// TIA Portal V19 export
FUNCTION "A0304_Navetta_CALL" : Void   // FC147, LAD
// stored: SetENOAutomatically false
BEGIN

REGION Network 1: <<< LATO TESTA >>>
END_REGION

REGION Network 2: DataIn - Ax
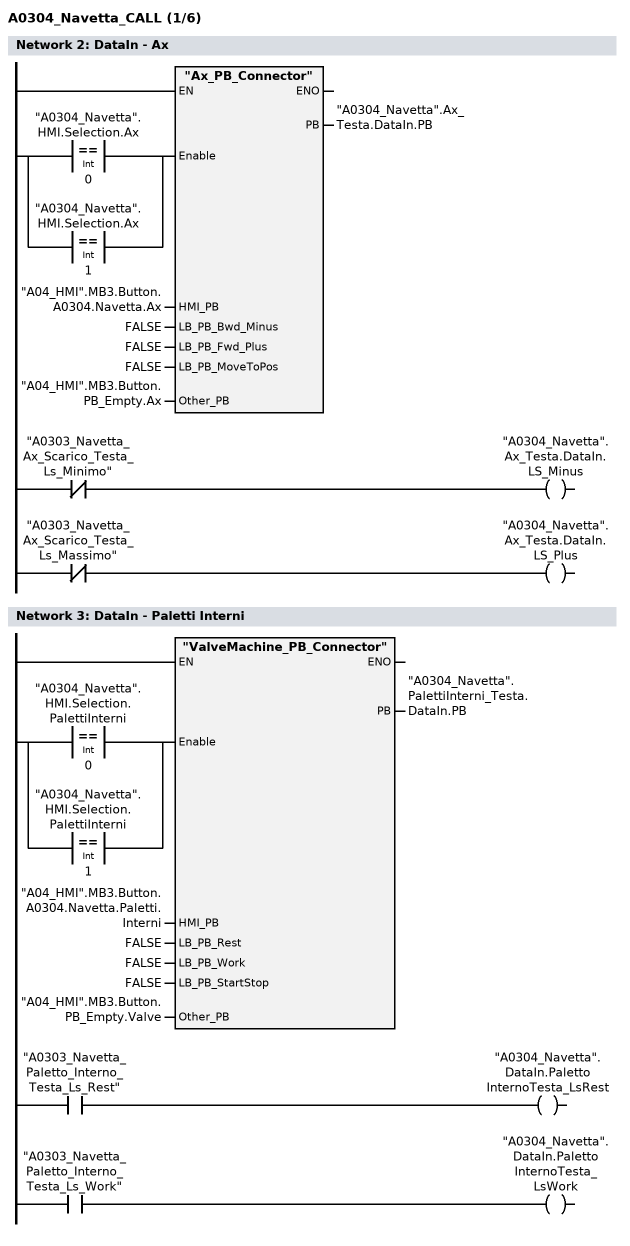
   RUNG wire#powerrail
      "Ax_PB_Connector"(Enable := wire#w1, HMI_PB := "A04_HMI".MB3.Button.A0304.Navetta.Ax, LB_PB_Bwd_Minus := FALSE, LB_PB_Fwd_Plus := FALSE, LB_PB_MoveToPos := FALSE, Other_PB := "A04_HMI".MB3.Button.PB_Empty.Ax, PB => "A0304_Navetta".Ax_Testa.DataIn.PB)
   END_RUNG
   RUNG wire#powerrail
      { S7_Templates := "SrcType := Int" } EQ_Contact(in1 := "A0304_Navetta".HMI.Selection.Ax, in2 := 0)
   END_RUNG wire#w1
   RUNG wire#powerrail
      { S7_Templates := "SrcType := Int" } EQ_Contact(in1 := "A0304_Navetta".HMI.Selection.Ax, in2 := 1)
   END_RUNG wire#w1
   RUNG wire#powerrail
      I_Contact( "A0303_Navetta_Ax_Scarico_Testa_Ls_Minimo" )
      Coil( "A0304_Navetta".Ax_Testa.DataIn.LS_Minus )
   END_RUNG
   RUNG wire#powerrail
      I_Contact( "A0303_Navetta_Ax_Scarico_Testa_Ls_Massimo" )
      Coil( "A0304_Navetta".Ax_Testa.DataIn.LS_Plus )
   END_RUNG
   // the same network as SCL:
   "Ax_PB_Connector"(Enable := ("A0304_Navetta".HMI.Selection.Ax = 0) OR ("A0304_Navetta".HMI.Selection.Ax = 1),
                     HMI_PB := "A04_HMI".MB3.Button.A0304.Navetta.Ax,
                     LB_PB_Bwd_Minus := FALSE,
                     LB_PB_Fwd_Plus := FALSE,
                     LB_PB_MoveToPos := FALSE,
                     Other_PB := "A04_HMI".MB3.Button.PB_Empty.Ax,
                     PB => "A0304_Navetta".Ax_Testa.DataIn.PB);
   "A0304_Navetta".Ax_Testa.DataIn.LS_Minus := NOT "A0303_Navetta_Ax_Scarico_Testa_Ls_Minimo";
   "A0304_Navetta".Ax_Testa.DataIn.LS_Plus := NOT "A0303_Navetta_Ax_Scarico_Testa_Ls_Massimo";
END_REGION

REGION Network 3: DataIn - Paletti Interni
   RUNG wire#powerrail
      "ValveMachine_PB_Connector"(Enable := wire#w1, HMI_PB := "A04_HMI".MB3.Button.A0304.Navetta.Paletti.Interni, LB_PB_Rest := FALSE, LB_PB_Work := FALSE, LB_PB_StartStop := FALSE, Other_PB := "A04_HMI".MB3.Button.PB_Empty.Valve, PB => "A0304_Navetta".PalettiInterni_Testa.DataIn.PB)
   END_RUNG
   RUNG wire#powerrail
      { S7_Templates := "SrcType := Int" } EQ_Contact(in1 := "A0304_Navetta".HMI.Selection.PalettiInterni, in2 := 0)
   END_RUNG wire#w1
   RUNG wire#powerrail
      { S7_Templates := "SrcType := Int" } EQ_Contact(in1 := "A0304_Navetta".HMI.Selection.PalettiInterni, in2 := 1)
   END_RUNG wire#w1
   RUNG wire#powerrail
      Contact( "A0303_Navetta_Paletto_Interno_Testa_Ls_Rest" )
      Coil( "A0304_Navetta".DataIn.PalettoInternoTesta_LsRest )
   END_RUNG
   RUNG wire#powerrail
      Contact( "A0303_Navetta_Paletto_Interno_Testa_Ls_Work" )
      Coil( "A0304_Navetta".DataIn.PalettoInternoTesta_LsWork )
   END_RUNG
   // the same network as SCL:
   "ValveMachine_PB_Connector"(Enable := ("A0304_Navetta".HMI.Selection.PalettiInterni = 0) OR ("A0304_Navetta".HMI.Selection.PalettiInterni = 1),
                           HMI_PB := "A04_HMI".MB3.Button.A0304.Navetta.Paletti.Interni,
                           LB_PB_Rest := FALSE,
                           LB_PB_Work := FALSE,
                           LB_PB_StartStop := FALSE,
                           Other_PB := "A04_HMI".MB3.Button.PB_Empty.Valve,
                           PB => "A0304_Navetta".PalettiInterni_Testa.DataIn.PB);
   "A0304_Navetta".DataIn.PalettoInternoTesta_LsRest := "A0303_Navetta_Paletto_Interno_Testa_Ls_Rest";
   "A0304_Navetta".DataIn.PalettoInternoTesta_LsWork := "A0303_Navetta_Paletto_Interno_Testa_Ls_Work";
END_REGION

REGION Network 4: DataIn - Paletti Esterni
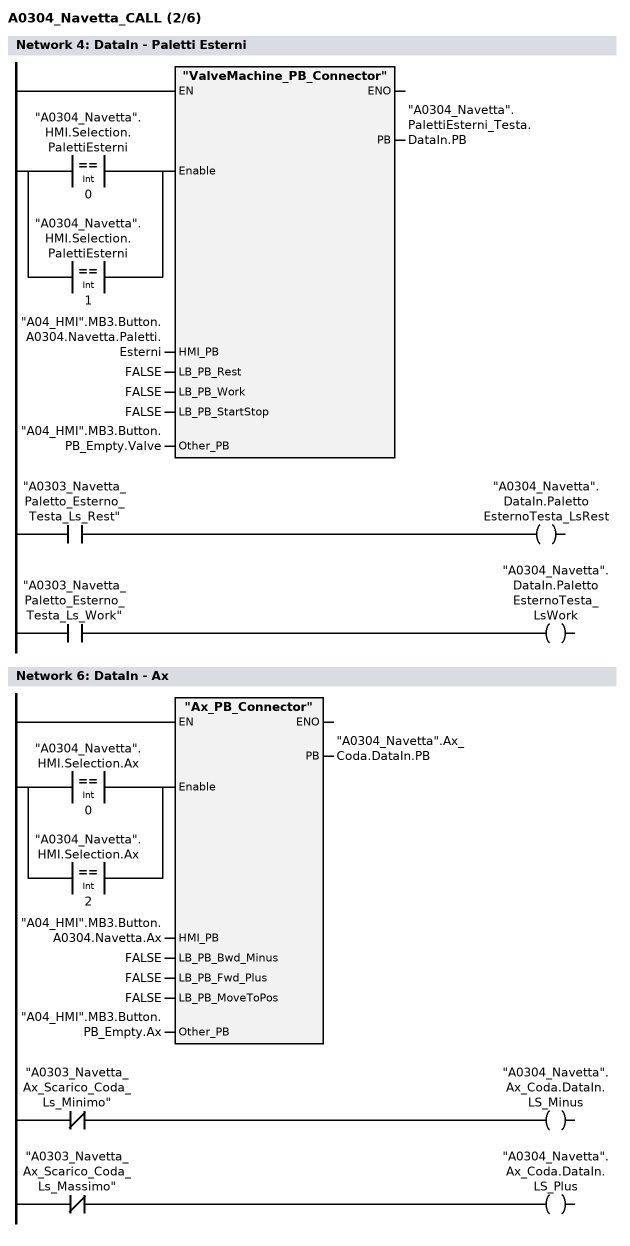
   RUNG wire#powerrail
      "ValveMachine_PB_Connector"(Enable := wire#w1, HMI_PB := "A04_HMI".MB3.Button.A0304.Navetta.Paletti.Esterni, LB_PB_Rest := FALSE, LB_PB_Work := FALSE, LB_PB_StartStop := FALSE, Other_PB := "A04_HMI".MB3.Button.PB_Empty.Valve, PB => "A0304_Navetta".PalettiEsterni_Testa.DataIn.PB)
   END_RUNG
   RUNG wire#powerrail
      { S7_Templates := "SrcType := Int" } EQ_Contact(in1 := "A0304_Navetta".HMI.Selection.PalettiEsterni, in2 := 0)
   END_RUNG wire#w1
   RUNG wire#powerrail
      { S7_Templates := "SrcType := Int" } EQ_Contact(in1 := "A0304_Navetta".HMI.Selection.PalettiEsterni, in2 := 1)
   END_RUNG wire#w1
   RUNG wire#powerrail
      Contact( "A0303_Navetta_Paletto_Esterno_Testa_Ls_Rest" )
      Coil( "A0304_Navetta".DataIn.PalettoEsternoTesta_LsRest )
   END_RUNG
   RUNG wire#powerrail
      Contact( "A0303_Navetta_Paletto_Esterno_Testa_Ls_Work" )
      Coil( "A0304_Navetta".DataIn.PalettoEsternoTesta_LsWork )
   END_RUNG
   // the same network as SCL:
   "ValveMachine_PB_Connector"(Enable := ("A0304_Navetta".HMI.Selection.PalettiEsterni = 0) OR ("A0304_Navetta".HMI.Selection.PalettiEsterni = 1),
                           HMI_PB := "A04_HMI".MB3.Button.A0304.Navetta.Paletti.Esterni,
                           LB_PB_Rest := FALSE,
                           LB_PB_Work := FALSE,
                           LB_PB_StartStop := FALSE,
                           Other_PB := "A04_HMI".MB3.Button.PB_Empty.Valve,
                           PB => "A0304_Navetta".PalettiEsterni_Testa.DataIn.PB);
   "A0304_Navetta".DataIn.PalettoEsternoTesta_LsRest := "A0303_Navetta_Paletto_Esterno_Testa_Ls_Rest";
   "A0304_Navetta".DataIn.PalettoEsternoTesta_LsWork := "A0303_Navetta_Paletto_Esterno_Testa_Ls_Work";
END_REGION

REGION Network 5: <<< LATO CODA >>>
END_REGION

REGION Network 6: DataIn - Ax
   RUNG wire#powerrail
      "Ax_PB_Connector"(Enable := wire#w1, HMI_PB := "A04_HMI".MB3.Button.A0304.Navetta.Ax, LB_PB_Bwd_Minus := FALSE, LB_PB_Fwd_Plus := FALSE, LB_PB_MoveToPos := FALSE, Other_PB := "A04_HMI".MB3.Button.PB_Empty.Ax, PB => "A0304_Navetta".Ax_Coda.DataIn.PB)
   END_RUNG
   RUNG wire#powerrail
      { S7_Templates := "SrcType := Int" } EQ_Contact(in1 := "A0304_Navetta".HMI.Selection.Ax, in2 := 0)
   END_RUNG wire#w1
   RUNG wire#powerrail
      { S7_Templates := "SrcType := Int" } EQ_Contact(in1 := "A0304_Navetta".HMI.Selection.Ax, in2 := 2)
   END_RUNG wire#w1
   RUNG wire#powerrail
      I_Contact( "A0303_Navetta_Ax_Scarico_Coda_Ls_Minimo" )
      Coil( "A0304_Navetta".Ax_Coda.DataIn.LS_Minus )
   END_RUNG
   RUNG wire#powerrail
      I_Contact( "A0303_Navetta_Ax_Scarico_Coda_Ls_Massimo" )
      Coil( "A0304_Navetta".Ax_Coda.DataIn.LS_Plus )
   END_RUNG
   // the same network as SCL:
   "Ax_PB_Connector"(Enable := ("A0304_Navetta".HMI.Selection.Ax = 0) OR ("A0304_Navetta".HMI.Selection.Ax = 2),
                     HMI_PB := "A04_HMI".MB3.Button.A0304.Navetta.Ax,
                     LB_PB_Bwd_Minus := FALSE,
                     LB_PB_Fwd_Plus := FALSE,
                     LB_PB_MoveToPos := FALSE,
                     Other_PB := "A04_HMI".MB3.Button.PB_Empty.Ax,
                     PB => "A0304_Navetta".Ax_Coda.DataIn.PB);
   "A0304_Navetta".Ax_Coda.DataIn.LS_Minus := NOT "A0303_Navetta_Ax_Scarico_Coda_Ls_Minimo";
   "A0304_Navetta".Ax_Coda.DataIn.LS_Plus := NOT "A0303_Navetta_Ax_Scarico_Coda_Ls_Massimo";
END_REGION

REGION Network 7: DataIn - Paletti Interni
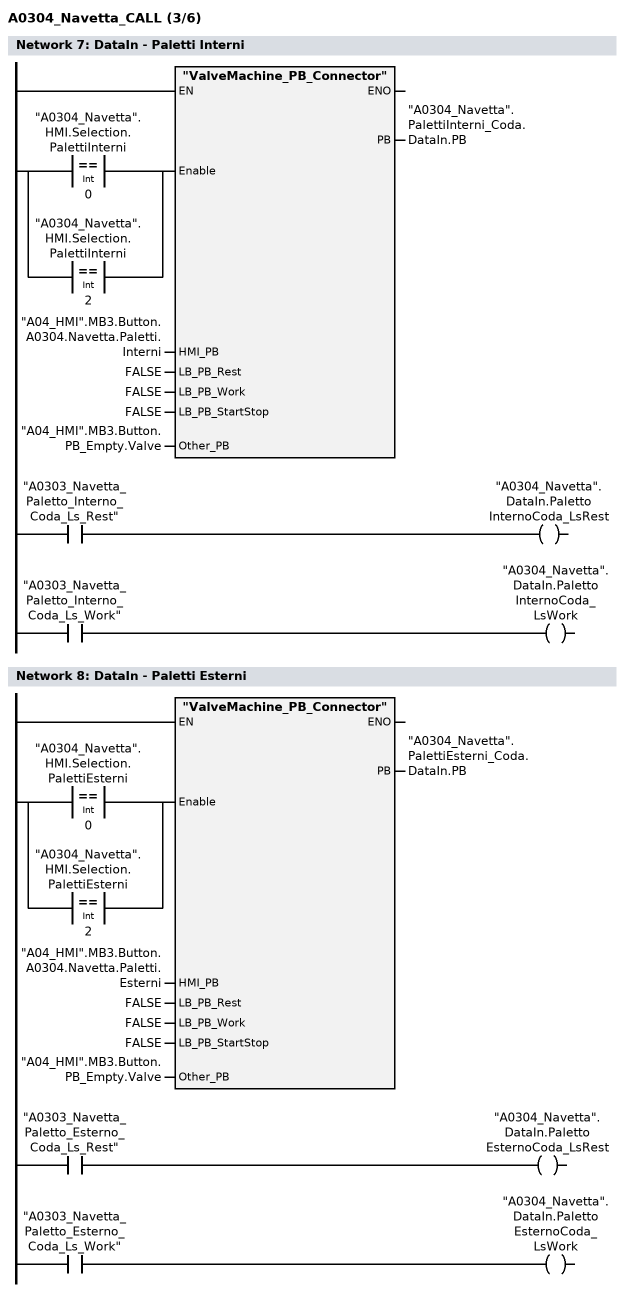
   RUNG wire#powerrail
      "ValveMachine_PB_Connector"(Enable := wire#w1, HMI_PB := "A04_HMI".MB3.Button.A0304.Navetta.Paletti.Interni, LB_PB_Rest := FALSE, LB_PB_Work := FALSE, LB_PB_StartStop := FALSE, Other_PB := "A04_HMI".MB3.Button.PB_Empty.Valve, PB => "A0304_Navetta".PalettiInterni_Coda.DataIn.PB)
   END_RUNG
   RUNG wire#powerrail
      { S7_Templates := "SrcType := Int" } EQ_Contact(in1 := "A0304_Navetta".HMI.Selection.PalettiInterni, in2 := 0)
   END_RUNG wire#w1
   RUNG wire#powerrail
      { S7_Templates := "SrcType := Int" } EQ_Contact(in1 := "A0304_Navetta".HMI.Selection.PalettiInterni, in2 := 2)
   END_RUNG wire#w1
   RUNG wire#powerrail
      Contact( "A0303_Navetta_Paletto_Interno_Coda_Ls_Rest" )
      Coil( "A0304_Navetta".DataIn.PalettoInternoCoda_LsRest )
   END_RUNG
   RUNG wire#powerrail
      Contact( "A0303_Navetta_Paletto_Interno_Coda_Ls_Work" )
      Coil( "A0304_Navetta".DataIn.PalettoInternoCoda_LsWork )
   END_RUNG
   // the same network as SCL:
   "ValveMachine_PB_Connector"(Enable := ("A0304_Navetta".HMI.Selection.PalettiInterni = 0) OR ("A0304_Navetta".HMI.Selection.PalettiInterni = 2),
                           HMI_PB := "A04_HMI".MB3.Button.A0304.Navetta.Paletti.Interni,
                           LB_PB_Rest := FALSE,
                           LB_PB_Work := FALSE,
                           LB_PB_StartStop := FALSE,
                           Other_PB := "A04_HMI".MB3.Button.PB_Empty.Valve,
                           PB => "A0304_Navetta".PalettiInterni_Coda.DataIn.PB);
   "A0304_Navetta".DataIn.PalettoInternoCoda_LsRest := "A0303_Navetta_Paletto_Interno_Coda_Ls_Rest";
   "A0304_Navetta".DataIn.PalettoInternoCoda_LsWork := "A0303_Navetta_Paletto_Interno_Coda_Ls_Work";
END_REGION

REGION Network 8: DataIn - Paletti Esterni
   RUNG wire#powerrail
      "ValveMachine_PB_Connector"(Enable := wire#w1, HMI_PB := "A04_HMI".MB3.Button.A0304.Navetta.Paletti.Esterni, LB_PB_Rest := FALSE, LB_PB_Work := FALSE, LB_PB_StartStop := FALSE, Other_PB := "A04_HMI".MB3.Button.PB_Empty.Valve, PB => "A0304_Navetta".PalettiEsterni_Coda.DataIn.PB)
   END_RUNG
   RUNG wire#powerrail
      { S7_Templates := "SrcType := Int" } EQ_Contact(in1 := "A0304_Navetta".HMI.Selection.PalettiEsterni, in2 := 0)
   END_RUNG wire#w1
   RUNG wire#powerrail
      { S7_Templates := "SrcType := Int" } EQ_Contact(in1 := "A0304_Navetta".HMI.Selection.PalettiEsterni, in2 := 2)
   END_RUNG wire#w1
   RUNG wire#powerrail
      Contact( "A0303_Navetta_Paletto_Esterno_Coda_Ls_Rest" )
      Coil( "A0304_Navetta".DataIn.PalettoEsternoCoda_LsRest )
   END_RUNG
   RUNG wire#powerrail
      Contact( "A0303_Navetta_Paletto_Esterno_Coda_Ls_Work" )
      Coil( "A0304_Navetta".DataIn.PalettoEsternoCoda_LsWork )
   END_RUNG
   // the same network as SCL:
   "ValveMachine_PB_Connector"(Enable := ("A0304_Navetta".HMI.Selection.PalettiEsterni = 0) OR ("A0304_Navetta".HMI.Selection.PalettiEsterni = 2),
                           HMI_PB := "A04_HMI".MB3.Button.A0304.Navetta.Paletti.Esterni,
                           LB_PB_Rest := FALSE,
                           LB_PB_Work := FALSE,
                           LB_PB_StartStop := FALSE,
                           Other_PB := "A04_HMI".MB3.Button.PB_Empty.Valve,
                           PB => "A0304_Navetta".PalettiEsterni_Coda.DataIn.PB);
   "A0304_Navetta".DataIn.PalettoEsternoCoda_LsRest := "A0303_Navetta_Paletto_Esterno_Coda_Ls_Rest";
   "A0304_Navetta".DataIn.PalettoEsternoCoda_LsWork := "A0303_Navetta_Paletto_Esterno_Coda_Ls_Work";
END_REGION

REGION Network 10: DataIn - Material Presence
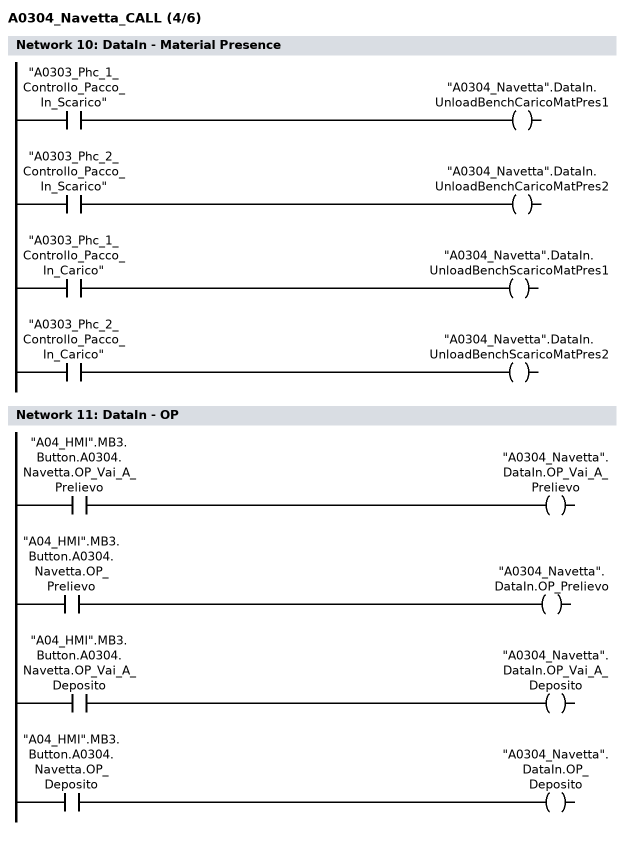
   RUNG wire#powerrail
      Contact( "A0303_Phc_1_Controllo_Pacco_In_Scarico" )
      Coil( "A0304_Navetta".DataIn.UnloadBenchCaricoMatPres1 )
   END_RUNG
   RUNG wire#powerrail
      Contact( "A0303_Phc_2_Controllo_Pacco_In_Scarico" )
      Coil( "A0304_Navetta".DataIn.UnloadBenchCaricoMatPres2 )
   END_RUNG
   RUNG wire#powerrail
      Contact( "A0303_Phc_1_Controllo_Pacco_In_Carico" )
      Coil( "A0304_Navetta".DataIn.UnloadBenchScaricoMatPres1 )
   END_RUNG
   RUNG wire#powerrail
      Contact( "A0303_Phc_2_Controllo_Pacco_In_Carico" )
      Coil( "A0304_Navetta".DataIn.UnloadBenchScaricoMatPres2 )
   END_RUNG
   // the same network as SCL:
   "A0304_Navetta".DataIn.UnloadBenchCaricoMatPres1 := "A0303_Phc_1_Controllo_Pacco_In_Scarico";
   "A0304_Navetta".DataIn.UnloadBenchCaricoMatPres2 := "A0303_Phc_2_Controllo_Pacco_In_Scarico";
   "A0304_Navetta".DataIn.UnloadBenchScaricoMatPres1 := "A0303_Phc_1_Controllo_Pacco_In_Carico";
   "A0304_Navetta".DataIn.UnloadBenchScaricoMatPres2 := "A0303_Phc_2_Controllo_Pacco_In_Carico";
END_REGION

REGION Network 11: DataIn - OP
   RUNG wire#powerrail
      Contact( "A04_HMI".MB3.Button.A0304.Navetta.OP_Vai_A_Prelievo )
      Coil( "A0304_Navetta".DataIn.OP_Vai_A_Prelievo )
   END_RUNG
   RUNG wire#powerrail
      Contact( "A04_HMI".MB3.Button.A0304.Navetta.OP_Prelievo )
      Coil( "A0304_Navetta".DataIn.OP_Prelievo )
   END_RUNG
   RUNG wire#powerrail
      Contact( "A04_HMI".MB3.Button.A0304.Navetta.OP_Vai_A_Deposito )
      Coil( "A0304_Navetta".DataIn.OP_Vai_A_Deposito )
   END_RUNG
   RUNG wire#powerrail
      Contact( "A04_HMI".MB3.Button.A0304.Navetta.OP_Deposito )
      Coil( "A0304_Navetta".DataIn.OP_Deposito )
   END_RUNG
   // the same network as SCL:
   "A0304_Navetta".DataIn.OP_Vai_A_Prelievo := "A04_HMI".MB3.Button.A0304.Navetta.OP_Vai_A_Prelievo;
   "A0304_Navetta".DataIn.OP_Prelievo := "A04_HMI".MB3.Button.A0304.Navetta.OP_Prelievo;
   "A0304_Navetta".DataIn.OP_Vai_A_Deposito := "A04_HMI".MB3.Button.A0304.Navetta.OP_Vai_A_Deposito;
   "A0304_Navetta".DataIn.OP_Deposito := "A04_HMI".MB3.Button.A0304.Navetta.OP_Deposito;
END_REGION

REGION Network 13: CIn
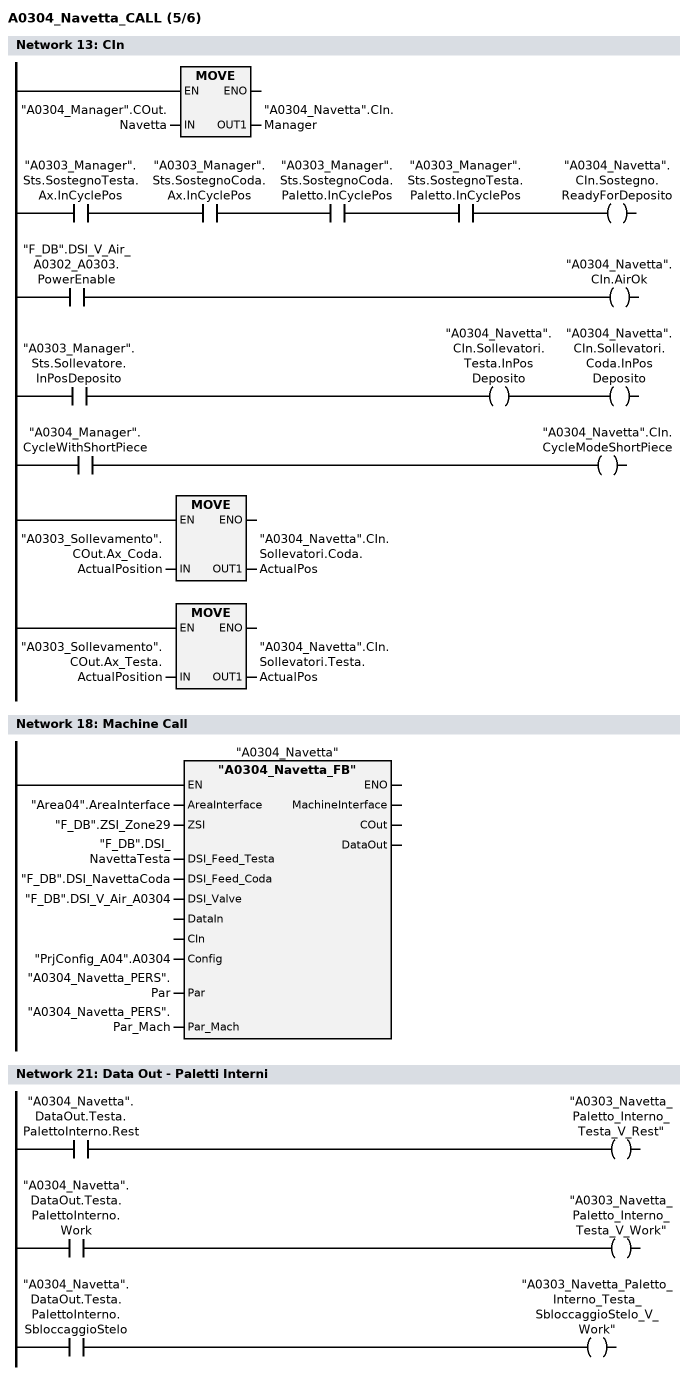
   RUNG wire#powerrail
      Move(in := "A0304_Manager".COut.Navetta, out1 => "A0304_Navetta".CIn.Manager)
   END_RUNG
   RUNG wire#powerrail
      Contact( "A0303_Manager".Sts.SostegnoTesta.Ax.InCyclePos )
      Contact( "A0303_Manager".Sts.SostegnoCoda.Ax.InCyclePos )
      Contact( "A0303_Manager".Sts.SostegnoCoda.Paletto.InCyclePos )
      Contact( "A0303_Manager".Sts.SostegnoTesta.Paletto.InCyclePos )
      Coil( "A0304_Navetta".CIn.Sostegno.ReadyForDeposito )
   END_RUNG
   RUNG wire#powerrail
      Contact( "F_DB".DSI_V_Air_A0302_A0303.PowerEnable )
      Coil( "A0304_Navetta".CIn.AirOk )
   END_RUNG
   RUNG wire#powerrail
      Contact( "A0303_Manager".Sts.Sollevatore.InPosDeposito )
      Coil( "A0304_Navetta".CIn.Sollevatori.Testa.InPosDeposito )
      Coil( "A0304_Navetta".CIn.Sollevatori.Coda.InPosDeposito )
   END_RUNG
   RUNG wire#powerrail
      Contact( "A0304_Manager".CycleWithShortPiece )
      Coil( "A0304_Navetta".CIn.CycleModeShortPiece )
   END_RUNG
   RUNG wire#powerrail
      Move(in := "A0303_Sollevamento".COut.Ax_Coda.ActualPosition, out1 => "A0304_Navetta".CIn.Sollevatori.Coda.ActualPos)
   END_RUNG
   RUNG wire#powerrail
      Move(in := "A0303_Sollevamento".COut.Ax_Testa.ActualPosition, out1 => "A0304_Navetta".CIn.Sollevatori.Testa.ActualPos)
   END_RUNG
   // the same network as SCL:
   "A0304_Navetta".CIn.Manager := "A0304_Manager".COut.Navetta;
   "A0304_Navetta".CIn.Sostegno.ReadyForDeposito := "A0303_Manager".Sts.SostegnoTesta.Ax.InCyclePos AND "A0303_Manager".Sts.SostegnoCoda.Ax.InCyclePos AND "A0303_Manager".Sts.SostegnoCoda.Paletto.InCyclePos AND "A0303_Manager".Sts.SostegnoTesta.Paletto.InCyclePos;
   "A0304_Navetta".CIn.AirOk := "F_DB".DSI_V_Air_A0302_A0303.PowerEnable;
   "A0304_Navetta".CIn.Sollevatori.Testa.InPosDeposito := "A0303_Manager".Sts.Sollevatore.InPosDeposito;
   "A0304_Navetta".CIn.Sollevatori.Coda.InPosDeposito := "A0303_Manager".Sts.Sollevatore.InPosDeposito;
   "A0304_Navetta".CIn.CycleModeShortPiece := "A0304_Manager".CycleWithShortPiece;
   "A0304_Navetta".CIn.Sollevatori.Coda.ActualPos := "A0303_Sollevamento".COut.Ax_Coda.ActualPosition;
   "A0304_Navetta".CIn.Sollevatori.Testa.ActualPos := "A0303_Sollevamento".COut.Ax_Testa.ActualPosition;
END_REGION

REGION Network 14: >
END_REGION

REGION Network 15 (SCL): Drive
   "A0304_Navetta".Ax_Testa.Drive.Infeed_ON := "Areas_ITF".AG.Infeed_Running;
   "A0304_Navetta".Ax_Testa.Drive.AccessPoint := "HW_Const_Values".CU8_PN_615A1_ModuleAccessPoint;
   "A0304_Navetta".Ax_Testa.Drive.AxisID := "CU8_ID_4_2430A1_1_2430M1";
   "A0304_Navetta".Ax_Testa.Drive.TokenChain := "TOKENCHAIN_CU8";

   "A0304_Navetta".Ax_Coda.Drive.Infeed_ON := "Areas_ITF".AG.Infeed_Running;
   "A0304_Navetta".Ax_Coda.Drive.AccessPoint := "HW_Const_Values".CU8_PN_615A1_ModuleAccessPoint;
   "A0304_Navetta".Ax_Coda.Drive.AxisID := "CU8_ID_5_2430A1_2_2460M1";
   "A0304_Navetta".Ax_Coda.Drive.TokenChain :=  "TOKENCHAIN_CU8";
END_REGION

REGION Network 16 (SCL): HW ID
   "A0304_Navetta".Ax_Testa.HW_ID_TEL1 := "HW_Const_Values".CU8_PN_2430A1_1_Standard_telegram_1;
   "A0304_Navetta".Enc_Testa.HW_IO := "HW_Const_Values".HW_2434P1_Telegram_81_DI_DO;

   "A0304_Navetta".Ax_Coda.HW_ID_TEL1 := "HW_Const_Values".CU8_PN_2430A1_2_Standard_telegram_1;
   "A0304_Navetta".Enc_Coda.HW_IO := "HW_Const_Values".HW_2464P1_Telegram_81_DI_DO;
END_REGION

REGION Network 17: >
END_REGION

REGION Network 18: Machine Call
   RUNG wire#powerrail
      "A0304_Navetta"(AreaInterface := "Area04".AreaInterface, ZSI := "F_DB".ZSI_Zone29, DSI_Feed_Testa := "F_DB".DSI_NavettaTesta, DSI_Feed_Coda := "F_DB".DSI_NavettaCoda, DSI_Valve := "F_DB".DSI_V_Air_A0304, DataIn :=, CIn :=, Config := "PrjConfig_A04".A0304, Par := "A0304_Navetta_PERS".Par, Par_Mach := "A0304_Navetta_PERS".Par_Mach, MachineInterface =>, COut =>, DataOut =>)
   END_RUNG
   // the same network as SCL:
   "A0304_Navetta"(AreaInterface := "Area04".AreaInterface,   // "A0304_Navetta_FB"
                   ZSI := "F_DB".ZSI_Zone29,
                   DSI_Feed_Testa := "F_DB".DSI_NavettaTesta,
                   DSI_Feed_Coda := "F_DB".DSI_NavettaCoda,
                   DSI_Valve := "F_DB".DSI_V_Air_A0304,
                   Config := "PrjConfig_A04".A0304,
                   Par := "A0304_Navetta_PERS".Par,
                   Par_Mach := "A0304_Navetta_PERS".Par_Mach);
END_REGION

REGION Network 20: <<< LATO TESTA >>>
END_REGION

REGION Network 21: Data Out - Paletti Interni
   RUNG wire#powerrail
      Contact( "A0304_Navetta".DataOut.Testa.PalettoInterno.Rest )
      Coil( "A0303_Navetta_Paletto_Interno_Testa_V_Rest" )
   END_RUNG
   RUNG wire#powerrail
      Contact( "A0304_Navetta".DataOut.Testa.PalettoInterno.Work )
      Coil( "A0303_Navetta_Paletto_Interno_Testa_V_Work" )
   END_RUNG
   RUNG wire#powerrail
      Contact( "A0304_Navetta".DataOut.Testa.PalettoInterno.SbloccaggioStelo )
      Coil( "A0303_Navetta_Paletto_Interno_Testa_SbloccaggioStelo_V_Work" )
   END_RUNG
   // the same network as SCL:
   "A0303_Navetta_Paletto_Interno_Testa_V_Rest" := "A0304_Navetta".DataOut.Testa.PalettoInterno.Rest;
   "A0303_Navetta_Paletto_Interno_Testa_V_Work" := "A0304_Navetta".DataOut.Testa.PalettoInterno.Work;
   "A0303_Navetta_Paletto_Interno_Testa_SbloccaggioStelo_V_Work" := "A0304_Navetta".DataOut.Testa.PalettoInterno.SbloccaggioStelo;
END_REGION

REGION Network 22: Data Out - Paletti Esterni
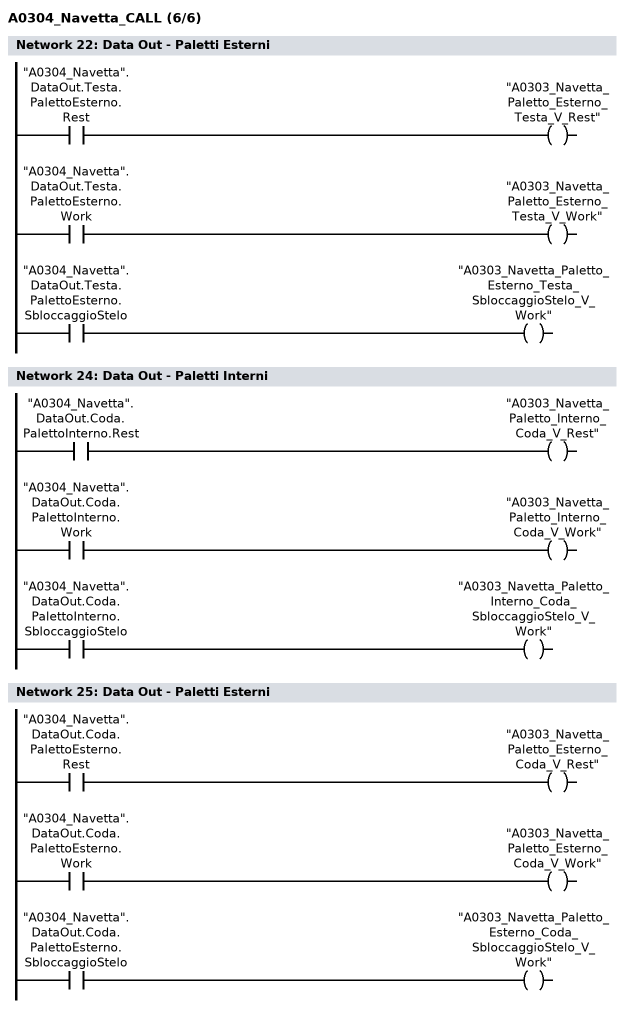
   RUNG wire#powerrail
      Contact( "A0304_Navetta".DataOut.Testa.PalettoEsterno.Rest )
      Coil( "A0303_Navetta_Paletto_Esterno_Testa_V_Rest" )
   END_RUNG
   RUNG wire#powerrail
      Contact( "A0304_Navetta".DataOut.Testa.PalettoEsterno.Work )
      Coil( "A0303_Navetta_Paletto_Esterno_Testa_V_Work" )
   END_RUNG
   RUNG wire#powerrail
      Contact( "A0304_Navetta".DataOut.Testa.PalettoEsterno.SbloccaggioStelo )
      Coil( "A0303_Navetta_Paletto_Esterno_Testa_SbloccaggioStelo_V_Work" )
   END_RUNG
   // the same network as SCL:
   "A0303_Navetta_Paletto_Esterno_Testa_V_Rest" := "A0304_Navetta".DataOut.Testa.PalettoEsterno.Rest;
   "A0303_Navetta_Paletto_Esterno_Testa_V_Work" := "A0304_Navetta".DataOut.Testa.PalettoEsterno.Work;
   "A0303_Navetta_Paletto_Esterno_Testa_SbloccaggioStelo_V_Work" := "A0304_Navetta".DataOut.Testa.PalettoEsterno.SbloccaggioStelo;
END_REGION

REGION Network 23: <<< LATO CODA >>>
END_REGION

REGION Network 24: Data Out - Paletti Interni
   RUNG wire#powerrail
      Contact( "A0304_Navetta".DataOut.Coda.PalettoInterno.Rest )
      Coil( "A0303_Navetta_Paletto_Interno_Coda_V_Rest" )
   END_RUNG
   RUNG wire#powerrail
      Contact( "A0304_Navetta".DataOut.Coda.PalettoInterno.Work )
      Coil( "A0303_Navetta_Paletto_Interno_Coda_V_Work" )
   END_RUNG
   RUNG wire#powerrail
      Contact( "A0304_Navetta".DataOut.Coda.PalettoInterno.SbloccaggioStelo )
      Coil( "A0303_Navetta_Paletto_Interno_Coda_SbloccaggioStelo_V_Work" )
   END_RUNG
   // the same network as SCL:
   "A0303_Navetta_Paletto_Interno_Coda_V_Rest" := "A0304_Navetta".DataOut.Coda.PalettoInterno.Rest;
   "A0303_Navetta_Paletto_Interno_Coda_V_Work" := "A0304_Navetta".DataOut.Coda.PalettoInterno.Work;
   "A0303_Navetta_Paletto_Interno_Coda_SbloccaggioStelo_V_Work" := "A0304_Navetta".DataOut.Coda.PalettoInterno.SbloccaggioStelo;
END_REGION

REGION Network 25: Data Out - Paletti Esterni
   RUNG wire#powerrail
      Contact( "A0304_Navetta".DataOut.Coda.PalettoEsterno.Rest )
      Coil( "A0303_Navetta_Paletto_Esterno_Coda_V_Rest" )
   END_RUNG
   RUNG wire#powerrail
      Contact( "A0304_Navetta".DataOut.Coda.PalettoEsterno.Work )
      Coil( "A0303_Navetta_Paletto_Esterno_Coda_V_Work" )
   END_RUNG
   RUNG wire#powerrail
      Contact( "A0304_Navetta".DataOut.Coda.PalettoEsterno.SbloccaggioStelo )
      Coil( "A0303_Navetta_Paletto_Esterno_Coda_SbloccaggioStelo_V_Work" )
   END_RUNG
   // the same network as SCL:
   "A0303_Navetta_Paletto_Esterno_Coda_V_Rest" := "A0304_Navetta".DataOut.Coda.PalettoEsterno.Rest;
   "A0303_Navetta_Paletto_Esterno_Coda_V_Work" := "A0304_Navetta".DataOut.Coda.PalettoEsterno.Work;
   "A0303_Navetta_Paletto_Esterno_Coda_SbloccaggioStelo_V_Work" := "A0304_Navetta".DataOut.Coda.PalettoEsterno.SbloccaggioStelo;
END_REGION
END_FUNCTION
